FUNCTION alg_s_Binitialized: BOOL
VAR_INPUT
    state: STATE;
END_VAR

alg_s_Binitialized := (state.dvar_M_HardwareMap) = (elit_initialized);

END_FUNCTION

(* stored: ProductVersion 3.1.0.18, Version 1.1.0.1 *)
